PROGRAM POU_writeReactorToSupvData
VAR
	sNetId: T_AmsNetId := SUPVams.sNetId;	// '5.30.23.91.1.1';
	nPort: T_AmsPort := SUPVams.nPort; 		// 851	

	FB_WriteAmsValue_XMEAS: FB_WriteAmsValue;
END_VAR

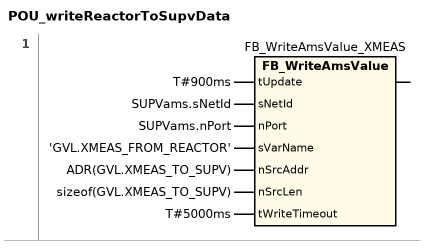
// NETWORK 1
FB_WriteAmsValue_XMEAS(
    tUpdate := T#900ms,
    sNetId := SUPVams.sNetId,
    nPort := SUPVams.nPort,
    sVarName := 'GVL.XMEAS_FROM_REACTOR',
    nSrcAddr := ADR(GVL.XMEAS_TO_SUPV),
    nSrcLen := sizeof(GVL.XMEAS_TO_SUPV),
    tWriteTimeout := T#5000ms); // FB_WriteAmsValue

END_PROGRAM

(* stored: Version 1.1.0.1, ProductVersion 3.1.4024.11
   POU POU_writeReactorToSupvData: Id {5e7ac2b2-7ed4-47ff-8a64-ec6be7ac94e9}, SpecialFunc None *)
